TYPE E_ProgramState : (
    PROGRAM_EMPTY := 0,
    PROGRAM_DRAFT := 10,
    PROGRAM_VALID := 20,
    PROGRAM_ACTIVE := 30,
    PROGRAM_INVALID := 40
); END_TYPE

(* stored: Version 1.1.0.1
   DUT E_ProgramState: Id {E3000000-0000-4000-8000-000000000025} *)
